{attribute 'GeneratedUsingTerminal: EK1122-0000-0018'}
{attribute addProperty BoxType "EK1122-0000-0018"}
{attribute addProperty Id "R10_AB00_EPP1322_0001R10_AB00_EPP1322_0001_481BC624168R10_AB1_EPP1008_0001EPP1008_78E8D3DD12R10_AB2_EPP1008_0001EPP1008_78E8D3DD12R10_AB3_EPP1008_0001EPP1008_78E8D3DD12R10_AB4_EPP1008_0001EPP1008_78E8D3DD12R10_AB5_EPP1008_0001EPP1008_78E8D3DD12R10_AB6_EPP1008_0001EPP1008_78E8D3DD12R10_AB02_EPP1332_0001EPP1332_1FC0878B2R10_AB7_EPP1008_0001EPP1008_78E8D3DD12R10_AB8_EPP1008_0001EPP1008_78E8D3DD12R10_AB11_EPP2308_0001EPP2308_F6D9A8D112R10_AB12_EPP2308_0001EPP2308_F6D9A8D112R10_AB13_EPP2308_0001EPP2308_F6D9A8D112"}
{attribute addProperty CRC "1780931621"}
{attribute addProperty Size "302"}
{attribute addProperty Name "R10_A3 (EK1122)"}
TYPE R10_A3_EK1122_6A26DC25 EXTENDS EK1122_1FC0878B : 
STRUCT
    {attribute addProperty Name "R10-AB00 (EPP1322-0001)"}
    {attribute addProperty PreviousPort "R10_A3 (EK1122) : D"}
    {attribute addProperty SyncUnit "default"}
    R10_AB00_EPP1322_0001 : R10_AB00_EPP1322_0001_481BC624;
    {attribute addProperty Name "R10-AB1 (EPP1008-0001)"}
    {attribute addProperty PreviousPort "R10-AB00 (EPP1322-0001) : C"}
    {attribute addProperty SyncUnit "R10"}
    R10_AB1_EPP1008_0001 : EPP1008_78E8D3DD;
    {attribute addProperty Name "R10-AB2 (EPP1008-0001)"}
    {attribute addProperty PreviousPort "R10-AB1 (EPP1008-0001) : B"}
    {attribute addProperty SyncUnit "R10"}
    R10_AB2_EPP1008_0001 : EPP1008_78E8D3DD;
    {attribute addProperty Name "R10-AB3 (EPP1008-0001)"}
    {attribute addProperty PreviousPort "R10-AB2 (EPP1008-0001) : B"}
    {attribute addProperty SyncUnit "R10"}
    R10_AB3_EPP1008_0001 : EPP1008_78E8D3DD;
    {attribute addProperty Name "R10-AB4 (EPP1008-0001)"}
    {attribute addProperty PreviousPort "R10-AB3 (EPP1008-0001) : B"}
    {attribute addProperty SyncUnit "R10"}
    R10_AB4_EPP1008_0001 : EPP1008_78E8D3DD;
    {attribute addProperty Name "R10-AB5 (EPP1008-0001)"}
    {attribute addProperty PreviousPort "R10-AB4 (EPP1008-0001) : B"}
    {attribute addProperty SyncUnit "R10"}
    R10_AB5_EPP1008_0001 : EPP1008_78E8D3DD;
    {attribute addProperty Name "R10-AB6 (EPP1008-0001)"}
    {attribute addProperty PreviousPort "R10-AB5 (EPP1008-0001) : B"}
    {attribute addProperty SyncUnit "R10"}
    R10_AB6_EPP1008_0001 : EPP1008_78E8D3DD;
    {attribute addProperty Name "R10-AB02 (EPP1332-0001)"}
    {attribute addProperty PreviousPort "R10-AB6 (EPP1008-0001) : B"}
    {attribute addProperty SyncUnit "default"}
    R10_AB02_EPP1332_0001 : EPP1332_1FC0878B;
    {attribute addProperty Name "R10-AB7 (EPP1008-0001)"}
    {attribute addProperty PreviousPort "R10-AB02 (EPP1332-0001) : C"}
    {attribute addProperty SyncUnit "R10"}
    R10_AB7_EPP1008_0001 : EPP1008_78E8D3DD;
    {attribute addProperty Name "R10-AB8 (EPP1008-0001)"}
    {attribute addProperty PreviousPort "R10-AB7 (EPP1008-0001) : B"}
    {attribute addProperty SyncUnit "R10"}
    R10_AB8_EPP1008_0001 : EPP1008_78E8D3DD;
    {attribute addProperty Name "R10-AB11 (EPP2308-0001)"}
    {attribute addProperty PreviousPort "R10-AB8 (EPP1008-0001) : B"}
    {attribute addProperty SyncUnit "R10"}
    R10_AB11_EPP2308_0001 : EPP2308_F6D9A8D1;
    {attribute addProperty Name "R10-AB12 (EPP2308-0001)"}
    {attribute addProperty PreviousPort "R10-AB11 (EPP2308-0001) : B"}
    {attribute addProperty SyncUnit "R10"}
    R10_AB12_EPP2308_0001 : EPP2308_F6D9A8D1;
    {attribute addProperty Name "R10-AB13 (EPP2308-0001)"}
    {attribute addProperty PreviousPort "R10-AB12 (EPP2308-0001) : B"}
    {attribute addProperty SyncUnit "R10"}
    R10_AB13_EPP2308_0001 : EPP2308_F6D9A8D1;
END_STRUCT
END_TYPE

(* stored: Version 1.2.0.0, ProductVersion 3.1.4024.11
   DUT R10_A3_EK1122_6A26DC25: Id {afe84994-f74c-0ecd-081a-1e05296bcd9b} *)
